Fanuc TP program (LS listing): B_AFLEG.LS

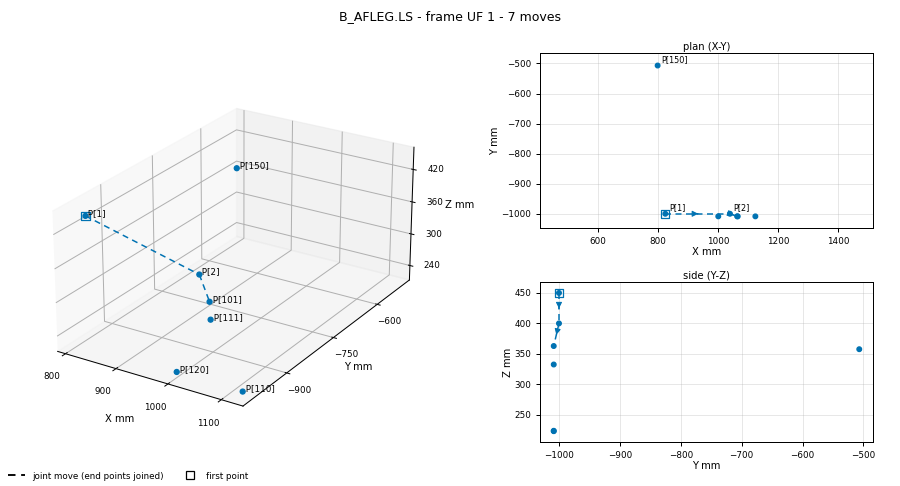
[picture p0: tool path of B_AFLEG.LS in frame UF 1, 7 of 11 moves have a stored position in this frame; points joined in program order, loops and branches not executed]
/PROG  B_AFLEG
/ATTR
OWNER		= MNEDITOR;
COMMENT		= "Afleg op corona";
PROG_SIZE	= 2163;
CREATE		= DATE 16-02-20  TIME 13:47:12;
MODIFIED	= DATE 19-01-22  TIME 18:30:56;
FILE_NAME	= AFLEGGEN;
VERSION		= 0;
LINE_COUNT	= 68;
MEMORY_SIZE	= 2699;
PROTECT		= READ_WRITE;
TCD:  STACK_SIZE	= 0,
      TASK_PRIORITY	= 50,
      TIME_SLICE	= 0,
      BUSY_LAMP_OFF	= 0,
      ABORT_REQUEST	= 0,
      PAUSE_REQUEST	= 0;
DEFAULT_GROUP	= 1,*,*,*,*;
CONTROL_CODE	= 00000000 00000000;
/APPL
/MN
   1:  DO[51:IONblower Corona]=ON ;
   2:   ;
   3:  UFRAME_NUM=1 ;
   4:  !Producten afleggen ;
   5:  !Wacht op afleg corona vry ;
   6:   ;
   7:  LBL[100:Start afleggen] ;
   8:  LBL[88:Draaien nar aflg] ;
   9:J P[1:Naar corona] 75% CNT50    ;
  10:J P[2:Boven corona] 75% CNT50    ;
  11:   ;
  12:  LBL[89] ;
  13:  !CHECK STORINGEN ;
  14:   ;
  15:  $WAITTMOUT=500 ;
  16:  WAIT DI[20:Afl 1 vrij Corona]=ON AND DI[21:Afl 2 vrij Corona]=ON TIMEOUT,LBL[200] ;
  17:   ;
  18:  IF DI[14:Tamponeren]=ON,JMP LBL[90] ;
  19:   ;
  20:  !Skinetta storing  ;
  21:  WAIT DI[93:FC uitloop vrij]=OFF TIMEOUT,LBL[200] ;
  22:   ;
  23:  !Pouch machine storing ;
  24:  WAIT DI[93:FC uitloop vrij]=OFF TIMEOUT,LBL[200] ;
  25:   ;
  26:  LBL[90] ;
  27:  DO[49:Buzzer hek]=OFF ;
  28:  DO[50:Rode lamp hek]=OFF ;
  29:   ;
  30:J P[101:Boven afleg ] 100% CNT30    ;
  31:  LBL[101] ;
  32:J P[110:AFLEG 2] 75% CNT50 Offset,PR[82:Boven afleg]    ;
  33:L P[110:AFLEG 2] 500mm/sec FINE    ;
  34:  Open hand 1    ;
  35:  WAIT    .25(sec) ;
  36:L P[110:AFLEG 2] 1000mm/sec CNT50 Offset,PR[82:Boven afleg]    ;
  37:   ;
  38:  IF R[21:Grijper 1-voudig]=1,JMP LBL[20] ;
  39:   ;
  40:J P[111:draaien] 75% CNT100 ACC50    ;
  41:   ;
  42:L P[120:AFLEG 1] 1000mm/sec CNT50 Offset,PR[82:Boven afleg]    ;
  43:L P[120:AFLEG 1] 500mm/sec FINE    ;
  44:  Open hand 2    ;
  45:  WAIT    .25(sec) ;
  46:L P[120:AFLEG 1] 650mm/sec CNT100 Offset,PR[82:Boven afleg]    ;
  47:   ;
  48:  LBL[20:1-VOUDIG] ;
  49:J P[150] 75% CNT100    ;
  50:   ;
  51:  IF R[9:Act R8]=0,JMP LBL[110] ;
  52:  IF R[9:Act R8]>=1 AND R[45:Teller ontstapel]=0,JMP LBL[210] ;
  53:   ;
  54:  JMP LBL[110] ;
  55:   ;
  56:  LBL[200:Buffer stapelen] ;
  57:  CALL BUF_STPL    ;
  58:  END ;
  59:   ;
  60:  LBL[210:Buffer leegmaken] ;
  61:  CALL BUF_ONTS    ;
  62:  IF R[42:Grijpfout bufffe]=1,JMP LBL[110] ;
  63:  JMP LBL[89] ;
  64:   ;
  65:  LBL[110:Einde programma] ;
  66:  R[45:Teller ontstapel]=0    ;
  67:  END ;
  68:   ;
/POS
P[1:"Naar corona"]{
   GP1:
	UF : 1, UT : 1,		CONFIG : 'F U T, 0, 0, 0',
	X =   825.000  mm,	Y = -1000.000  mm,	Z =   450.000  mm,
	W =   -89.915 deg,	P =      .505 deg,	R =   179.664 deg
};
P[2:"Boven corona"]{
   GP1:
	UF : 1, UT : 1,		CONFIG : 'N U T, 0, 0, 0',
	X =  1040.000  mm,	Y = -1000.000  mm,	Z =   400.000  mm,
	W =   179.747 deg,	P =     -.806 deg,	R =   -92.046 deg
};
P[101:"Boven afleg "]{
   GP1:
	UF : 1, UT : 1,		CONFIG : 'N U T, 0, 0, 0',
	X =  1064.127  mm,	Y = -1008.616  mm,	Z =   362.822  mm,
	W =   179.662 deg,	P =      .062 deg,	R =   -92.024 deg
};
P[110:"AFLEG 2"]{
   GP1:
	UF : 1, UT : 1,		CONFIG : 'N U T, 0, 0, 0',
	X =  1124.607  mm,	Y = -1008.616  mm,	Z =   222.966  mm,
	W =   179.662 deg,	P =      .062 deg,	R =   -92.024 deg
};
P[111:"draaien"]{
   GP1:
	UF : 1, UT : 1,		CONFIG : 'N U T, 0, 0, 0',
	X =  1065.855  mm,	Y = -1008.615  mm,	Z =   332.485  mm,
	W =   179.662 deg,	P =      .062 deg,	R =   -38.430 deg
};
P[120:"AFLEG 1"]{
   GP1:
	UF : 1, UT : 1,		CONFIG : 'N U T, 0, 0, 0',
	X =  1001.227  mm,	Y = -1008.615  mm,	Z =   223.676  mm,
	W =   179.662 deg,	P =      .062 deg,	R =    88.499 deg
};
P[150]{
   GP1:
	UF : 1, UT : 1,		CONFIG : 'N U T, 0, 0, 0',
	X =   799.479  mm,	Y =  -506.909  mm,	Z =   357.592  mm,
	W =   179.538 deg,	P =      .252 deg,	R =    -1.191 deg
};
/END
